
// ===== library: MasterCopy "Calculo_mm" =====

FUNCTION "Calculo_mm" : Void   // FC1, SCL
{ S7_Optimized_Access := 'TRUE' }
VERSION : 0.1
   VAR_INPUT
      Lectura_pulsos : DInt;
      Radio : Real;
      Resolucion_encoder : Int;
   END_VAR
   VAR_OUTPUT
      mm_recorridos : Real;
   END_VAR
   VAR CONSTANT
      pi : Real := 3.1415;
   END_VAR
BEGIN
   #mm_recorridos := (#Lectura_pulsos * #Radio * 2 * #pi) / #Resolucion_encoder;
END_FUNCTION

// ===== library: MasterCopy "Analog_IN" =====

FUNCTION_BLOCK "Analog_IN"   // FB4, LAD
{ S7_Optimized_Access := 'TRUE' }
VERSION : 0.1
   VAR_INPUT
      Input : Int;
      X_min : Real;
      X_max : Real;
      Y_min : Real;
      Y_max : Real;
      IsTension : Bool;
   END_VAR
   VAR_OUTPUT
      Output : Real;
   END_VAR
   VAR
      X_min_bits : Int;
      X_max_bits : Int;
      norm : Real;
   END_VAR
   VAR CONSTANT
      tension_pendent : Real := 2764.8;
      intensity_pendent : Real := 1382.4;
   END_VAR
BEGIN

REGION Network 1 (SCL)

   IF #IsTension THEN
       #X_min_bits := REAL_TO_INT(#X_min * #tension_pendent);
       #X_max_bits := REAL_TO_INT(#X_max * #tension_pendent);
   ELSE
       #X_min_bits := REAL_TO_INT(#X_min * #intensity_pendent);
       #X_max_bits := REAL_TO_INT(#X_max * #intensity_pendent);
   END_IF;
END_REGION

REGION Network 2
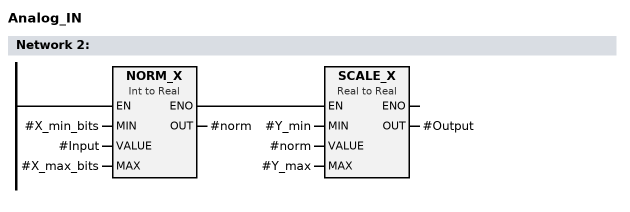
   RUNG wire#powerrail
      { S7_Templates := "[SrcType := Int, DestType := Real]" } Normalize(min := #X_min_bits, value := #Input, max := #X_max_bits, out => #norm)
      { S7_Templates := "[SrcType := Real, DestType := Real]" } Scale(min := #Y_min, value := #norm, max := #Y_max, out => #Output)
   END_RUNG
   // the same network as SCL:
   #norm := NORM_X(MIN := #X_min_bits, VALUE := #Input, MAX := #X_max_bits);
   #Output := SCALE_X(MIN := #Y_min, VALUE := #norm, MAX := #Y_max);
END_REGION
END_FUNCTION_BLOCK

// ===== library: MasterCopy "Analog_OUT" =====

FUNCTION_BLOCK "Analog_OUT"   // FB5, LAD
{ S7_Optimized_Access := 'TRUE' }
VERSION : 0.1
   VAR_INPUT
      Input : Real;
      X_min : Real;
      X_max : Real;
      Y_min : Real;
      Y_max : Real;
      IsTension : Bool;
   END_VAR
   VAR_OUTPUT
      Output : Int;
   END_VAR
   VAR
      Y_min_bits : Int;
      Y_max_bits : Int;
      norm : Real;
   END_VAR
   VAR CONSTANT
      tension_pendent : Real := 2764.8;
      intensity_pendent : Real := 1382.4;
   END_VAR
BEGIN

REGION Network 1 (SCL)

   IF #IsTension THEN
       #Y_min_bits := REAL_TO_INT(#Y_min * #tension_pendent);
       #Y_max_bits := REAL_TO_INT(#Y_max * #tension_pendent);
   ELSE
       #Y_min_bits := REAL_TO_INT(#Y_min * #intensity_pendent);
       #Y_max_bits := REAL_TO_INT(#Y_max * #intensity_pendent);
   END_IF;
END_REGION

REGION Network 2
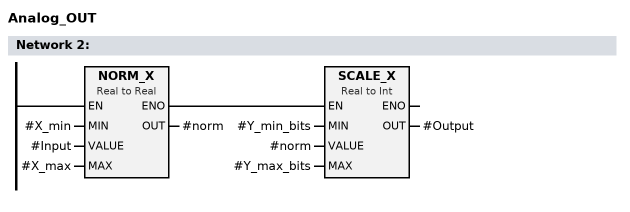
   RUNG wire#powerrail
      { S7_Templates := "[SrcType := Real, DestType := Real]" } Normalize(min := #X_min, value := #Input, max := #X_max, out => #norm)
      { S7_Templates := "[SrcType := Real, DestType := Int]" } Scale(min := #Y_min_bits, value := #norm, max := #Y_max_bits, out => #Output)
   END_RUNG
   // the same network as SCL:
   #norm := NORM_X(MIN := #X_min, VALUE := #Input, MAX := #X_max);
   #Output := SCALE_X(MIN := #Y_min_bits, VALUE := #norm, MAX := #Y_max_bits);
END_REGION
END_FUNCTION_BLOCK

// ===== library: MasterCopy "Arranque_EstTri" =====

FUNCTION_BLOCK "Arranque_EstTri"   // FB3, LAD
{ S7_Optimized_Access := 'TRUE' }
VERSION : 0.1
   VAR_INPUT
      Tiempo : Time;
      Start : Bool;
      Stop : Bool;
   END_VAR
   VAR_OUTPUT
      Línea : Bool;
      Estrella : Bool;
      Triángulo : Bool;
   END_VAR
   VAR
      temporizador_1 : IEC_TIMER;
      IEC_Timer_0_Instance : TON_TIME;
   END_VAR
BEGIN

REGION Network 1
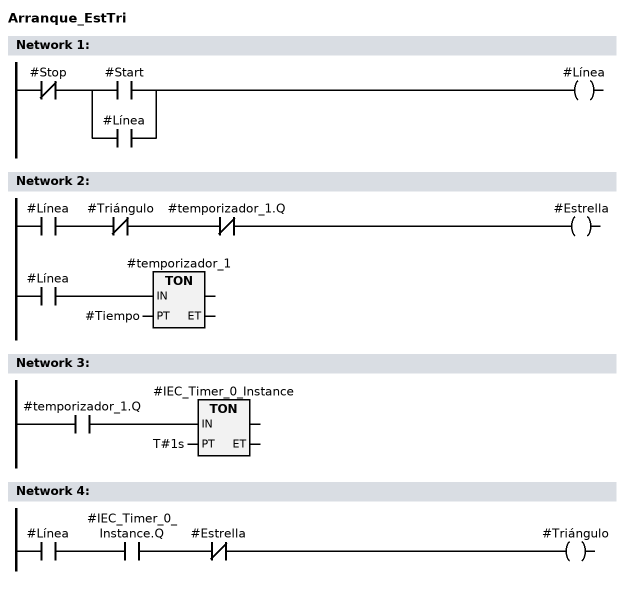
   RUNG wire#powerrail
      I_Contact( #Stop )
      wire#w1
      Contact( #Start )
      wire#w2
      Coil( #Línea )
   END_RUNG
   RUNG wire#w1
      Contact( #Línea )
   END_RUNG wire#w2
   // the same network as SCL:
   #Línea := NOT #Stop AND (#Start OR #Línea);
END_REGION

REGION Network 2
   #Estrella := #Línea AND NOT #Triángulo AND NOT #temporizador_1.Q;
   #temporizador_1.TON(IN := #Línea, PT := #Tiempo);
END_REGION

REGION Network 3
   #IEC_Timer_0_Instance(IN := #temporizador_1.Q, PT := T#1s);   // TON
END_REGION

REGION Network 4
   RUNG wire#powerrail
      Contact( #Línea )
      Contact( #IEC_Timer_0_Instance.Q )
      I_Contact( #Estrella )
      Coil( #Triángulo )
   END_RUNG
   // the same network as SCL:
   #Triángulo := #Línea AND #IEC_Timer_0_Instance.Q AND NOT #Estrella;
END_REGION
END_FUNCTION_BLOCK

// ===== library: MasterCopy "Calculo_milimetros" =====

FUNCTION_BLOCK "Calculo_milimetros"   // FB1, SCL
{ S7_Optimized_Access := 'TRUE' }
VERSION : 0.1
   VAR_INPUT
      Lectura_pulsos : DInt;
      Radio : Real;
      Resolucion_encoder : Int;
   END_VAR
   VAR_OUTPUT
      mm_recorridos : Real;
   END_VAR
   VAR CONSTANT
      pi : Real := 3.1415;
   END_VAR
BEGIN
   #mm_recorridos := (#Lectura_pulsos * #Radio * 2 * #pi) / #Resolucion_encoder;
END_FUNCTION_BLOCK

// ===== library: MasterCopy "Telerruptor" =====

FUNCTION_BLOCK "Telerruptor"   // FB2, LAD
{ S7_Optimized_Access := 'TRUE' }
VERSION : 0.1
   VAR_INPUT
      Pulsador : Bool;
   END_VAR
   VAR_OUTPUT
      Salida : Bool;
   END_VAR
   VAR
      Flanco : Bool;
      "on/off" : Bool;
      state : Bool;
   END_VAR
   VAR_TEMP   // added for the SCL form of the ladder/FBD networks
      _w1 : Bool;
   END_VAR
BEGIN

REGION Network 1
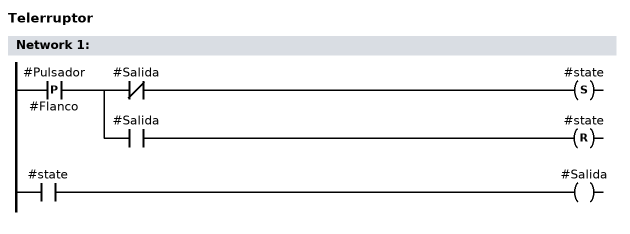
   RUNG wire#powerrail
      P_Contact(operand := #Pulsador, bit := #Flanco)
      wire#w1
      I_Contact( #Salida )
      S_Coil( #state )
   END_RUNG
   RUNG wire#w1
      Contact( #Salida )
      R_Coil( #state )
   END_RUNG
   RUNG wire#powerrail
      Contact( #state )
      Coil( #Salida )
   END_RUNG
   // the same network as SCL:
   #_w1 := #Pulsador AND NOT #Flanco;   // rising edge of #Pulsador
   #Flanco := #Pulsador;
   IF #_w1 AND NOT #Salida THEN #state := TRUE; END_IF;
   IF #_w1 AND #Salida THEN #state := FALSE; END_IF;
   #Salida := #state;
END_REGION
END_FUNCTION_BLOCK